           10:  // Set Calibration activ?
               IF "gtyp_Setup".x_Color_Sensor_Calibration
                   AND ("gtyp_Setup".i_Color_Sensor_Selection = 1) THEN
                   "gtyp_Setup".x_Calculate_Value_Color := FALSE;
                   "gtyp_Setup".x_Set_Calib_Value_Color_Blue := FALSE;
                   "gtyp_Setup".x_Set_Calib_Value_Color_Red := FALSE;
                   "gtyp_Setup".x_Set_Calib_Value_Color_White := FALSE;
                   "gtyp_Setup".w_Calib_ColorValue_Blue := 0;
                   "gtyp_Setup".w_Calib_ColorValue_Red := 0;
                   "gtyp_Setup".w_Calib_ColorValue_White := 0;
                   "gtyp_Setup".w_Threshold_Red_Blue := 0;
                   "gtyp_Setup".w_Threshold_White_Red := 0;
                   #li_StepCase := 20;
               END_IF;

           20: // wait for set Values or Calculate

               // Start new Positioning
               IF "gtyp_Setup".x_Set_Calib_Value_Color_Blue THEN
                   "gtyp_Setup".w_Calib_ColorValue_Blue := "IW_SSC_ColorSensor_A1";
                   "gtyp_Setup".x_Set_Calib_Value_Color_Blue := FALSE;
               ELSIF "gtyp_Setup".x_Set_Calib_Value_Color_Red THEN
                   "gtyp_Setup".w_Calib_ColorValue_Red := "IW_SSC_ColorSensor_A1";
                   "gtyp_Setup".x_Set_Calib_Value_Color_Red := FALSE;
               ELSIF "gtyp_Setup".x_Set_Calib_Value_Color_White THEN
                   "gtyp_Setup".w_Calib_ColorValue_White := "IW_SSC_ColorSensor_A1";
                   "gtyp_Setup".x_Set_Calib_Value_Color_White := FALSE;
               END_IF;

               "gtyp_Setup".w_Threshold_White_Red  := "gtyp_Setup".w_Calib_ColorValue_White + (("gtyp_Setup".w_Calib_ColorValue_Red - "gtyp_Setup".w_Calib_ColorValue_White) / 2);
               "gtyp_Setup".w_Threshold_Red_Blue   := "gtyp_Setup".w_Calib_ColorValue_Red + (("gtyp_Setup".w_Calib_ColorValue_Blue - "gtyp_Setup".w_Calib_ColorValue_Red) / 2);

               IF "gtyp_Setup".x_Calculate_Value_Color THEN
                   "gtyp_SSC".w_Threshold_White_Red := "gtyp_Setup".w_Threshold_White_Red;
                   "gtyp_SSC".w_Threshold_Red_Blue := "gtyp_Setup".w_Threshold_Red_Blue;
                   "gtyp_Setup".x_Calculate_Value_Color := FALSE;
               END_IF;

               // Statement section ELSE    
           ELSE
               ;
       END_CASE;

       IF ("gtyp_Setup".i_Color_Sensor_Selection = 1) THEN
           // Reload Pos Value
           "gtyp_Setup".w_Actual_ColorValue := "IW_SSC_ColorSensor_A1";
       END_IF;
   ELSE
       #lx_Init := TRUE;
   END_IF;
END_FUNCTION_BLOCK

FUNCTION_BLOCK "PRG_DSO_Status"   // FB36, SCL
TITLE = Program Status DSO
{ S7_Optimized_Access := 'TRUE' }
AUTHOR : A.Schaefer
VERSION : 0.0
   VAR
      lx_Init : Bool;
      lx_Start : Bool;
      li_StepCase : Int;
      ldt_MQTT : Date_And_Time;
      li_Return_LDT : Int;
      li_code_old : Int;
      lfb_R_Trig_Outsourcing : R_TRIG;
      lfb_R_Trig_Take_Workpiece : R_TRIG;
      lfb_TON_Status : TON_TIME;
      lfb_TON_End_Order : TON_TIME;
      lx_StartStatus : Bool;
      lx_StartEndOrder : Bool;
      lx_StartTimer : Bool;
   END_VAR
BEGIN
   IF #lx_Init THEN

       // wait time state
       #lfb_TON_Status(IN := NOT #lx_StartStatus,
                       PT := T#2s);

       // rising/falling edge light barrier DSI
       #lfb_R_Trig_Outsourcing(CLK := NOT "IX_SSC_LightBarrierOutsourcing_I4");
       #lfb_R_Trig_Take_Workpiece(CLK := "IX_SSC_LightBarrierOutsourcing_I4");

       // start wait time end order 
       IF NOT "IX_SSC_LightBarrierOutsourcing_I4" AND ("gtyp_Interface_Dashboard".Subscribe.State_Order.s_state = 'SHIPPED') THEN
           #lx_StartEndOrder := TRUE;
       END_IF;

       // wait time end order
       #lfb_TON_End_Order(IN := #lx_StartEndOrder,
                          PT := T#5s);

       IF #lfb_R_Trig_Take_Workpiece.Q OR #lfb_TON_End_Order.Q THEN
           #lx_StartEndOrder := FALSE;
           "gtyp_Interface_Dashboard".Subscribe.State_Order.ldt_ts := DT_TO_LDT(#ldt_MQTT);
           "gtyp_Interface_Dashboard".Subscribe.State_Order.s_state := 'WAITING_FOR_ORDER';
           "gtyp_Interface_Dashboard".Subscribe.State_Order.s_type := '';
           "gtyp_Interface_Dashboard".Subscribe.State_DSO.x_active := FALSE;
       END_IF;

       // state of the DSO transmitted to the cloud
       IF (#lfb_TON_Status.Q OR #lfb_R_Trig_Outsourcing.Q OR #lfb_R_Trig_Take_Workpiece.Q) AND NOT #lx_StartStatus THEN
           #lx_StartStatus := TRUE;
           #li_Return_LDT := RD_SYS_T(#ldt_MQTT);
           IF NOT "IX_SSC_LightBarrierOutsourcing_I4" THEN
               "gtyp_Interface_Dashboard".Subscribe.State_DSO.i_code := 0;
           ELSE
               "gtyp_Interface_Dashboard".Subscribe.State_DSO.i_code := 1;
           END_IF;
           "gtyp_Interface_Dashboard".Subscribe.State_DSO.ldt_ts := DT_TO_LDT(#ldt_MQTT);
           "gtyp_Interface_Dashboard".Subscribe.State_DSO.s_station := 'dso';
           "gtyp_Interface_Dashboard".Subscribe.State_DSO.s_target := '';
           "gtyp_Interface_Dashboard".Subscribe.State_DSO.s_description := '';
       END_IF;

       IF NOT #lfb_TON_Status.Q AND #lx_StartStatus THEN
           #lx_StartStatus := FALSE;
       END_IF;
   ELSE
       #lx_Init := TRUE;
       #lx_StartEndOrder := FALSE;
   END_IF;
END_FUNCTION_BLOCK

FUNCTION_BLOCK "PRG_DSI_Status"   // FB37, SCL
TITLE = Program Status DSI
{ S7_Optimized_Access := 'TRUE' }
AUTHOR : A.Schaefer
VERSION : 0.0
   VAR
      lx_Init : Bool;
      lx_Start : Bool;
      li_StepCase : Int;
      ldt_MQTT : Date_And_Time;
      li_Return_LDT : Int;
      lfb_R_Trig_Storage : R_TRIG;
      lfb_F_Trig_Storage : F_TRIG;
      lfb_TON_Status : TON_TIME;
      lx_StartStatus : Bool;
      lfb_TON_Schritt : TON_TIME;
      lx_StartTimer : Bool;
   END_VAR
BEGIN
   IF #lx_Init THEN

       // wait time state
       #lfb_TON_Status(IN := NOT #lx_StartStatus,
                       PT := T#2s);

       // rising/falling edge light barrier DSI
       #lfb_R_Trig_Storage(CLK := NOT "IX_SSC_LightBarrierStorage_I3");
       #lfb_F_Trig_Storage(CLK := NOT "IX_SSC_LightBarrierStorage_I3");

       // state of the DSI transmitted to the cloud
       IF (#lfb_TON_Status.Q OR #lfb_R_Trig_Storage.Q OR #lfb_F_Trig_Storage.Q) AND NOT #lx_StartStatus THEN
           #lx_StartStatus := TRUE;
           #li_Return_LDT := RD_SYS_T(#ldt_MQTT);
           IF NOT "IX_SSC_LightBarrierStorage_I3" THEN
               "gtyp_Interface_Dashboard".Subscribe.State_DSI.i_code := 0;
               "gtyp_Interface_Dashboard".Subscribe.State_DSI.x_active := TRUE;
           ELSE
               "gtyp_Interface_Dashboard".Subscribe.State_DSI.i_code := 1;
               IF #lfb_F_Trig_Storage.Q THEN
                   "gtyp_Interface_Dashboard".Subscribe.State_DSI.x_active := FALSE;
               END_IF;
           END_IF;
           "gtyp_Interface_Dashboard".Subscribe.State_DSI.ldt_ts := DT_TO_LDT(#ldt_MQTT);
           "gtyp_Interface_Dashboard".Subscribe.State_DSI.s_station := 'dsi';
           "gtyp_Interface_Dashboard".Subscribe.State_DSI.s_target := '';
           "gtyp_Interface_Dashboard".Subscribe.State_DSI.s_description := '';
       END_IF;

       IF NOT #lfb_TON_Status.Q AND #lx_StartStatus THEN
           #lx_StartStatus := FALSE;
       END_IF;
   ELSE
       #lx_Init := TRUE;
   END_IF;
END_FUNCTION_BLOCK